FUNCTION TryConvert_UINT_TO_LREAL : BOOL
VAR_INPUT
	in : UINT;
	out : REFERENCE TO LREAL;
END_VAR

out := UINT_TO_LREAL(in);
TryConvert_UINT_TO_LREAL := TRUE;

END_FUNCTION

(* stored: Version 1.1.0.1, ProductVersion 3.1.4024.12
   POU TryConvert_UINT_TO_LREAL: Id {70df9f66-7d94-4eaa-9780-10a3f3f776ae}, SpecialFunc None *)
